INTERFACE EventLogger

METHOD logEvent : BOOL
VAR_INPUT
END_VAR
END_METHOD

METHOD queueEvent : BOOL
VAR_INPUT
	event : INT;
END_VAR
END_METHOD

END_INTERFACE

(* stored: Version 1.1.0.1, ProductVersion 3.1.4024.11
   Itf EventLogger: Id {2533d092-9fe0-4b9a-8fe9-ea815fba24a7}
   Method logEvent: Id {ee387f80-b4ac-4ea1-bc00-7527cdf4a3ce}
   Method queueEvent: Id {7850d4f0-b066-45f5-a717-807658f58f81} *)
